// TIA Portal V16 export
// export: Created 2024-12-03T15:41:42.8061657Z, ExportSetting WithDefaults, DisplayName Totally Integrated Automation Portal, DisplayVersion V16 Update 6, DisplayName TIA Portal Version Control Interface, DisplayVersion V16 Update 2, DisplayName TIA Portal Openness, DisplayVersion V16 Update 6, DisplayName TIA Portal Teamcenter Gateway, DisplayVersion V16, DisplayName SINAMICS Startdrive Advanced, DisplayVersion V16 Update 5, DisplayName SINAMICS Startdrive G130, G150, S120, S150, SINAMICS MV, S210, DisplayVersion V16 Update 5, DisplayName SINAMICS Startdrive G110M, G120, G120C, G120D, G120P, G115D, DisplayVersion V16 Update 5, DisplayName STEP 7 Professional, DisplayVersion V16 Update 6, DisplayName STEP 7 Safety, DisplayVersion V16, DisplayName WinCC Advanced / Unified PC, DisplayVersion V16 Update 6
FUNCTION_BLOCK "Motor_DOL_Controller_FB"   // FB69, SCL
{ S7_Optimized_Access := 'TRUE' }
VERSION : 0.1
// stored: AutoNumber true, IsIECCheckEnabled false, IsRetainMemResEnabled false, MemoryReserve 100, SetENOAutomatically false, UDAEnableTagReadback false
   VAR_INPUT
      I_Interlock : Bool;
      I_RunningFeedBack : Bool;
      I_ThermalProtection : Bool;
      I_TimeNotRunning : Time := t#10s;
      I_TimeNotStopping : Time := t#10s;
      I_TimeRunningFeedbackDelay : Time;
   END_VAR
   VAR_OUTPUT
      O_CmdOn : Bool;
      O_CmdDirection : Bool;
   END_VAR
   VAR_IN_OUT
      IO_Motor : "Motor_DOL_UDT";
   END_VAR
   VAR DB_SPECIFIC
      S_TimeNotRunning { S7_SetPoint := 'True'} : TON_TIME;
      S_TimeNotStopping { S7_SetPoint := 'True'} : TON_TIME;
      S_TimeRunningFeedBack { S7_SetPoint := 'True'} : TON_TIME;
   END_VAR
   VAR
      info { S7_SetPoint := 'True'} : "AlarmInfo_UDT";
   END_VAR
   VAR_TEMP
      T_ZoneInfo : "ZoneInfo";
      T_AppState : "ApplicationState_UDT";
   END_VAR
BEGIN
   #T_ZoneInfo := "ApplicationState_DB".ZoneNames[#IO_Motor.Zone];
   #T_AppState := "ApplicationState_DB".Appstate[#T_ZoneInfo.AppStateIndex];
   REGION Copy commands

       #IO_Motor.Status.ManualCommandsDisabled := 0;
       #O_CmdDirection := false;
       #O_CmdOn := false;

       //Auto mode
       IF "ApplicationState_DB".Appstate[#IO_Motor.Zone].States.AutoModeActivated.State THEN
           #O_CmdOn := #IO_Motor.Cmd.OnAuto;
           #O_CmdDirection := #IO_Motor.Cmd.DirectionAuto;
       END_IF;

       //Turn commands of if manual mode is deactivated
       IF NOT "ApplicationState_DB".Appstate[#IO_Motor.Zone].States.ManualModeActivated.State OR
           #IO_Motor.Alarms.AlarmStatus > 0 OR
           NOT "ApplicationState_DB".Appstate[#IO_Motor.Zone].States.EmergencyOk.State
           OR #IO_Motor.Status.Interlocked THEN
           #IO_Motor.Cmd.OnManual := 0;
           #IO_Motor.Cmd.DirectionManual := 0;
           #IO_Motor.Status.ManualCommandsDisabled := 1;
       END_IF;

       //Manual mode
       IF "ApplicationState_DB".Appstate[#IO_Motor.Zone].States.ManualModeActivated.State THEN
           #O_CmdOn := #IO_Motor.Cmd.OnManual := #IO_Motor.Cmd.OnManual;
           #O_CmdDirection := #IO_Motor.Cmd.DirectionManual;
       END_IF;

   END_REGION

   REGION Interlock

       #IO_Motor.Status.Interlocked := #I_Interlock OR #IO_Motor.Cmd.Interlock;
       #IO_Motor.Status.Status.%X0 := #IO_Motor.Status.Interlocked;

   END_REGION

   REGION Manual MODe active

       #IO_Motor.Status.ManualModeActive := "ApplicationState_DB".Appstate[#IO_Motor.Zone].States.ManualModeActivated.State;
       #IO_Motor.Status.Status.%X2 := #IO_Motor.Status.ManualModeActive;

   END_REGION

   REGION Turn commands off on error

       IF #IO_Motor.Alarms.AlarmStatus > 0
           OR NOT "ApplicationState_DB".Appstate[#IO_Motor.Zone].States.EmergencyOk.State
           OR #IO_Motor.Status.Interlocked THEN
           #O_CmdOn := 0;
       END_IF;

   END_REGION

   REGION INFO
       IF NOT #info.init OR #IO_Motor.Name = '' THEN
           #IO_Motor.Name := "buildObjectName"(I_Symbolname := GetSymbolName(variable := #IO_Motor, size := 100));
           #info.info := "buildAlarmInfo"(I_ObjectName := #IO_Motor.Name, I_ZoneIndex := #IO_Motor.Zone, I_ZoneName := #T_ZoneInfo.ZoneName);
           #info.init := true;
       END_IF;
   END_REGION

   REGION alarms

       #S_TimeNotRunning(IN := #O_CmdOn AND NOT #IO_Motor.Status.Running,
                         PT := t#10s);

       IF #S_TimeNotRunning.Q THEN
           #IO_Motor.Alarms.NotOnTImedOut.Active := true;
       END_IF;

       #S_TimeNotStopping(IN := NOT #O_CmdOn AND #IO_Motor.Status.Running,
                          PT := t#10s);

       IF #S_TimeNotStopping.Q THEN
           #IO_Motor.Alarms.NotOffTimedOut.Active := TRUE;
           #IO_Motor.Alarms.NotOffTimedOut.Active := FALSE;
       END_IF;

       IF NOT #I_ThermalProtection THEN
           #IO_Motor.Alarms.ThermalProtection.Active := true;
       END_IF;

       IF #IO_Motor.Alarms.AlarmStatus > 0 THEN
           "ApplicationState_DB".Appstate[#T_ZoneInfo.AppStateIndex].Alarms.AlarmActiveInternalPLC := TRUE;
       END_IF;

   END_REGION

   REGION Create alarm status

       #IO_Motor.Alarms.AlarmStatus.%X0 := #IO_Motor.Alarms.NotOnTImedOut.Active;
       #IO_Motor.Alarms.AlarmStatus.%X1 := #IO_Motor.Alarms.NotOffTimedOut.Active;
       #IO_Motor.Alarms.AlarmStatus.%X2 := #IO_Motor.Alarms.ThermalProtection.Active;

   END_REGION

   REGION Reset 

       IF #T_AppState.Hmi_Buttons.reset.state.State
           OR #IO_Motor.Cmd.Reset THEN
           #IO_Motor.Alarms.ThermalProtection.Active := 0;
           #IO_Motor.Alarms.NotOffTimedOut.Active := 0;
           #IO_Motor.Alarms.NotOnTImedOut.Active := 0;
       END_IF;

   END_REGION

   REGION Running feedback

       #S_TimeRunningFeedBack(IN:=#I_RunningFeedBack,
                              PT:=#I_TimeRunningFeedbackDelay,
                              Q=>#IO_Motor.Status.Running);

       #IO_Motor.Status.Status.%X1 := #IO_Motor.Status.Running;

   END_REGION

   REGION Create common status

       #IO_Motor.CommonStatus := 0;
       IF #IO_Motor.Status.Running THEN
           #IO_Motor.CommonStatus:= 1;
       END_IF;

       IF #IO_Motor.Alarms.AlarmStatus > 1 THEN
           #IO_Motor.CommonStatus := 2;
       END_IF;

   END_REGION

   #IO_Motor.Cmd.Reset := 0;
END_FUNCTION_BLOCK
